# EPICS autosave request: soft_iocs/galil_DMC_E03/iocBoot/iocgalil_DMC_E03/GalilTest_18ID_DMC_E03Positions.req
$(P)17.DVAL
$(P)18.DVAL
$(P)19.DVAL
$(P)20.DVAL
$(P)21.DVAL
$(P)22.DVAL
$(P)23.DVAL
$(P)24.DVAL
